INTERFACE I_ForwardEnumerator EXTENDS I_Disposable

PROPERTY PUBLIC IsValid : BOOL
GET
END_GET
END_PROPERTY

METHOD PUBLIC MoveNext : BOOL
END_METHOD

METHOD PUBLIC Reset
END_METHOD

METHOD PUBLIC TryGet : BOOL;
VAR_INPUT
    Destination : ANY;
END_VAR
END_METHOD

METHOD PUBLIC TryGetTo : BOOL;
VAR_INPUT
    DestinationAddress : PVOID;
    DestinationSize : UDINT;
END_VAR
END_METHOD

END_INTERFACE

(* stored: Version 1.1.0.1, ProductVersion 3.1.4024.12
   Itf I_ForwardEnumerator: Id {54058b9b-80fc-4e81-9e5f-09690cd78563}
   Property IsValid: Id {774b7fb2-3ab9-415f-afbd-38b67c12c836}
   Get Get: Id {1b31618a-c412-471c-aa32-94a098218a3b}
   Method MoveNext: Id {2f1007bb-2d3b-422e-8363-1ac17138fff6}
   Method Reset: Id {9832dfa1-60c0-02b4-201c-8f38260263fa}
   Method TryGet: Id {e3ad555a-1ec0-4e33-ad3b-b4fe6907ee09}
   Method TryGetTo: Id {b0bb221f-cc0b-40e9-b0f6-6bb61f735c6a} *)
